PROGRAM VerkeersLichtR
VAR
	HuidigeStatus : VerkeerslichtStatus := VerkeerslichtStatus.Rood; //Start met rood
    Timer1 : TON; 
END_VAR


IF GVL.AutoR THEN //Als er een auto bij het stoplicht staat (de knop naast de lichten)
    CASE HuidigeStatus OF
        VerkeerslichtStatus.Rood:
            Timer1(IN := TRUE, PT := GVL.TijdRood);
            IF Timer1.Q THEN
                HuidigeStatus := VeranderLicht(HuidigeStatus);
                Timer1(IN := FALSE);
				
				GVL.GroenR := FALSE;
            	GVL.GeelR := FALSE;
            	GVL.RoodR := TRUE;   // Zet Rood licht aan

            END_IF
        VerkeerslichtStatus.Groen:
            Timer1(IN := TRUE, PT := GVL.TijdGroen);
            IF Timer1.Q THEN
                HuidigeStatus := VeranderLicht(HuidigeStatus);
                Timer1(IN := FALSE);
				
				GVL.GroenR := TRUE;   // Zet Groen licht aan
            	GVL.GeelR := FALSE;
           		GVL.RoodR := FALSE;
				
            END_IF
        VerkeerslichtStatus.Geel:
            Timer1(IN := TRUE, PT := GVL.TijdGeel);
            IF Timer1.Q THEN
                HuidigeStatus := VeranderLicht(HuidigeStatus);
                Timer1(IN := FALSE);
				
				GVL.GroenR := FALSE;
           		GVL.GeelR := TRUE;    // Zet Geel licht aan
            	GVL.RoodR := FALSE;
            END_IF
    END_CASE
ELSE
    // Als er geen auto aankomt, gaat het verkeerslicht op rood
    HuidigeStatus := VerkeerslichtStatus.Rood;
    GVL.GroenR := FALSE;
    GVL.GeelR := FALSE;
    GVL.RoodR := TRUE;
END_IF

GVL.LichtStatusR := HuidigeStatus; // Dit zorgt ervoor dat de GVL wordt ge-update

END_PROGRAM

(* stored: Version 1.1.0.1, ProductVersion 3.1.4024.12
   POU VerkeersLichtR: Id {6b3d4ad0-f3f9-4c2c-9fe5-74f1d2e9b24b}, SpecialFunc None *)
